FUNCTION_BLOCK FB_HardwareInit
VAR_INPUT
    bExecute : BOOL;  // Command to start the motors initialization
    bReset   : BOOL;  // Command to reset the FB state
END_VAR

VAR_OUTPUT
    bDone  : BOOL;  // Indicates that initialization was completed successfully
    bError : BOOL;  // Indicates an error in the process
END_VAR

VAR
    bMoveAxis    : BOOL := FALSE;
    bMoveServo   : BOOL := FALSE;
    
    fbResetM1, fbResetM2, fbResetM3 : FB_MotorsReset;
    fbMotorsPowerUp : FB_MotorsPowerUp;
    bPowerUp    : BOOL := FALSE;
    
    fbHomeM1, fbHomeM2, fbHomeM3 : FB_HomePosition;
    fbMoveValves : ARRAY[1..5] OF FB_ValvePositionControl;
    TonPowerUp : TON;
    
    iState : INT := -1; // Default state is reset (-1)
	i	   : INT; //loop for index

    // Event Logger Variables
    fbEventHandler : FB_EventHandler;
    fbEventTrigger : R_TRIG;  // Event Trigger
    bExecuteEvent  : BOOL := FALSE;
    bEventDone     : BOOL := FALSE;
END_VAR

CASE iState OF

    // State -1: Reset state
    -1:
        bDone := FALSE;
        bError := FALSE;
        bMoveAxis := FALSE;
        bMoveServo := FALSE;
        bExecuteEvent := FALSE;
        bEventDone := FALSE;
		fbResetM1.Reset();
		fbResetM2.Reset();
		fbResetM3.Reset();
		
        
        // Ensure all motors and actuators are reset
        //GVL_Safety.bAirSupplyEnable := FALSE;
        //GVL_Safety.bDoorLockCommand := FALSE;

        IF bExecute AND NOT bReset THEN
            iState := 0; // Proceed to initialization
        END_IF;

    // State 0: Reset motors before enabling them
    0: 
        fbResetM1(bExecute := bExecute, Axis := GVL_Motion.M1Motor.Axis);
        fbResetM2(bExecute := bExecute, Axis := GVL_Motion.M2Motor.Axis);
        fbResetM3(bExecute := bExecute, Axis := GVL_Motion.M3Motor.Axis);

        IF fbResetM1.bDone AND fbResetM2.bDone AND fbResetM3.bDone THEN
            iState := 1;
        END_IF;
        
        IF fbResetM1.bError OR fbResetM2.bError OR fbResetM3.bError THEN
            iState := 99;
        END_IF;

    // State 1: Power up the motors
    1:
        fbMotorsPowerUp(bExecute := TRUE);
        
        IF fbMotorsPowerUp.bPowerUpDone THEN
            iState := 2; // Next step
        END_IF;
        
    // State 2: Homing Motors M1 -> M2
    2:
        bError := FALSE;
        bMoveAxis := bExecute;

        TonPowerUp(IN := TRUE, PT := T#2S); // Time necessary to power up the motors before moving them
        
        IF TonPowerUp.Q AND NOT fbHomeM1.bHomingDone AND NOT fbHomeM1.bError THEN
            fbHomeM1(eMotor := E_Motors.M1StageCollection, bStartHoming := bMoveAxis);
        END_IF;
        
        IF TonPowerUp.Q AND NOT fbHomeM2.bHomingDone AND NOT fbHomeM2.bError THEN
            fbHomeM2(eMotor := E_Motors.M2SampleRecVertical, bStartHoming := bMoveAxis);
        END_IF;
        
        // If homing was done, next state
        IF fbHomeM1.bHomingDone AND fbHomeM2.bHomingDone THEN
            iState := 3;
        END_IF;

        // If there is an error in M1 or M2, stop the process
        IF fbHomeM1.bError OR fbHomeM2.bError THEN
            iState := 99;
        END_IF;

    // State 3: Homing M3
    3:
        IF NOT fbHomeM3.bHomingDone AND NOT fbHomeM3.bError THEN
            fbHomeM3(eMotor := E_Motors.M3SampleRecHorizontal, bStartHoming := bMoveAxis);
        END_IF;

        IF fbHomeM3.bHomingDone AND NOT fbHomeM3.bError THEN
            bMoveAxis := FALSE;
            iState := 4;
        END_IF;

        IF fbHomeM3.bError THEN
            bError := TRUE;
            iState := 99;
        END_IF;

    // State 4: Move valves to home position
    4:
        bMoveServo := bExecute;
		//TODO - M6 Valve 4 motor is damage and because of that was taken out of the logic to keep working until it is replaced
		(*FOR i := 1 TO 3 DO
        	fbMoveValves[i](bEnable := bMoveServo, ServoAxis := GVL_Motion.aValves[i].Axis, iValvePosition := 1);
        END_FOR
		*)
		fbMoveValves[1](bEnable := bMoveServo, ServoAxis := GVL_Motion.aValves[1].Axis, iValvePosition := 1);
		fbMoveValves[2](bEnable := bMoveServo, ServoAxis := GVL_Motion.aValves[2].Axis, iValvePosition := 1);
		fbMoveValves[4](bEnable := bMoveServo, ServoAxis := GVL_Motion.aValves[4].Axis, iValvePosition := 1);
		fbMoveValves[5](bEnable := bMoveServo, ServoAxis := GVL_Motion.aValves[5].Axis, iValvePosition := 1);
		
		
        // Check if all servos have reached home position
        IF fbMoveValves[1].bMoveDone AND fbMoveValves[2].bMoveDone (* AND fbMoveValves[3].bMoveDone *) AND fbMoveValves[4].bMoveDone AND fbMoveValves[5].bMoveDone THEN
            bDone := TRUE;
            bMoveServo := FALSE;
            iState := 100; // End State
        END_IF;
        
        // Check if any servo has an error
        IF fbMoveValves[1].bError OR fbMoveValves[2].bError (* OR fbMoveValves[3].bError *) OR fbMoveValves[4].bError OR fbMoveValves[5].bError  THEN
            bError := TRUE;
            iState := 99;
        END_IF;

    // State 99: Error State
    99:
        bError := TRUE;
        bDone := FALSE;
        bMoveAxis := FALSE;
        bMoveServo := FALSE;
        
        // Event Logger error message
        bExecuteEvent := TRUE;
        fbEventTrigger(CLK := bExecuteEvent);
        IF fbEventTrigger.Q THEN
            fbEventHandler(bExecute:= TRUE, eEventName:= E_Events.ERROR, sSystem:= 'Hardware Init', sMessage:= 'Initialization Failed!', bDone=> bEventDone);
        END_IF;

    // State 100: Hardware Init Completed
    100:
        // Event Logger success message
        bExecuteEvent := TRUE;
        IF NOT bEventDone THEN
            fbEventHandler(bExecute := bExecuteEvent, eEventName := E_Events.INFO, sSystem := 'Hardware Init', sMessage := 'Hardware Initialized Successfully!', bDone => bEventDone);
        END_IF;
        bExecuteEvent := FALSE;
        bDone := TRUE;
        
        // Reset state machine if reset is triggered
        IF bReset THEN
            iState := -1;
        END_IF;

END_CASE;

METHOD Reset : BOOL
VAR_INPUT
END_VAR
END_METHOD

ACTION ResetEventTrigger:
IF bEventDone THEN
        bExecuteEvent := FALSE;
        bEventDone := FALSE;
END_IF;
END_ACTION

END_FUNCTION_BLOCK

(* stored: Version 1.1.0.1, ProductVersion 3.1.4024.12
   POU FB_HardwareInit: Id {31780309-bb82-4307-91d5-5548f242181e}, SpecialFunc None
   Method Reset: Id {18d6fe1a-c7c5-4df1-bb63-009c872ad55c}
   Action ResetEventTrigger: Id {49b081fb-821b-4506-a920-a26eb4c501f1} *)
